{attribute 'GeneratedUsingTerminal: EL2212-0000-0018'}
{attribute addProperty BoxType "EL2212-0000-0018"}
{attribute addProperty Id "ControlAT %Q*Control_4E83000D3"}
{attribute addProperty CRC "2806981475"}
{attribute addProperty Size "3"}
TYPE DOX_Control_Channel_A74F2363 :
STRUCT
	{attribute addProperty Name "Control"}
	Control AT %Q* : Control_4E83000D;
END_STRUCT
END_TYPE

(* stored: Version 1.2.0.0, ProductVersion 3.1.4024.9
   DUT DOX_Control_Channel_A74F2363: Id {e5aa9c1c-2544-466f-a060-3f759cabb347} *)
